# EPICS substitutions: evrSupport/Db/ioc/bsaPMTEdef.substitutions
#==============================================================================
#
# Abs:  Beam Synchronous Acquisition records for a single
#	photo multiplier tube (PMT).
#
# Name: bsaPMTEdef.substitutions
#
# Note: Must follow the LCLS naming conventions.
#
#==============================================================================
#
file bsaATTREdef.db
{
#           Device   Attribute  Input            EGU     HOPR  LOPR PREC ADEL  Link
  pattern {   D       , ATTR ,   I             , EG    ,  HO  , LO , PR , AD ,  LNK,     SINK_SIZE  }
	  { $(DEVICE) ,QDCRAW, $(DEVICE):QDCRAW, count , 65535, 0  ,  3 ,  1 , $(SLCLNK), $(SINK_SIZE\=10) }
}
